// TIA Portal V17 export
// export: Created 2024-09-02T12:50:20.1310188Z, ExportSetting WithDefaults, DisplayName Totally Integrated Automation Portal, DisplayVersion V17, DisplayName TIA Portal Openness, DisplayVersion V17, DisplayName TIA Portal Version Control Interface, DisplayVersion V17, DisplayName STEP 7 Professional, DisplayVersion V17, DisplayName STEP 7 Safety, DisplayVersion V17, DisplayName WinCC Professional, DisplayVersion V17
FUNCTION "AnwFC3_FG02_Saving_Status_SLG3_OP70" : Void   // FC1113, LAD
TITLE = Recalculate Moby / Rückberechnen Moby
{ S7_Optimized_Access := 'TRUE' }
AUTHOR : OlegFuehrus
FAMILY : MOBY
NAME : OlegFuehrus
VERSION : 0.1
// stored: AutoNumber false, IsIECCheckEnabled false, SetENOAutomatically false, UDAEnableTagReadback false
   VAR_TEMP
      t_VKE0 : Bool;   // VKE0
      t_VKE1 : Bool;   // VKE1
      t_Melderk_IO : Bool;   // Meldekontrollen SOLL==IST / Reporting controls SOLL==IST
      t_Status : Byte;   // Bearbeitungstatus / Processing status
      t_TafNr : Int;   // Aktuelle TAF Nummer / Current TAF number
      t_BeaNr : Int;   // Aktuelle BEA Nummer / Current BEA number
      t_END : Bool;
      Save_IO : Bool;
      Save_IO_1 : Bool;
   END_VAR
   VAR CONSTANT
      konst_kennung_schrauber : Byte := 31;
      konst_kennung_fuegen : Byte := 42;
      konst_kennung_wegmessung : Byte := 45;
      konst_kennung_reibmoment : Byte := 46;
      konst_kennung_losbrechmoment : Byte := 47;
   END_VAR
BEGIN

REGION Network 1: INIT
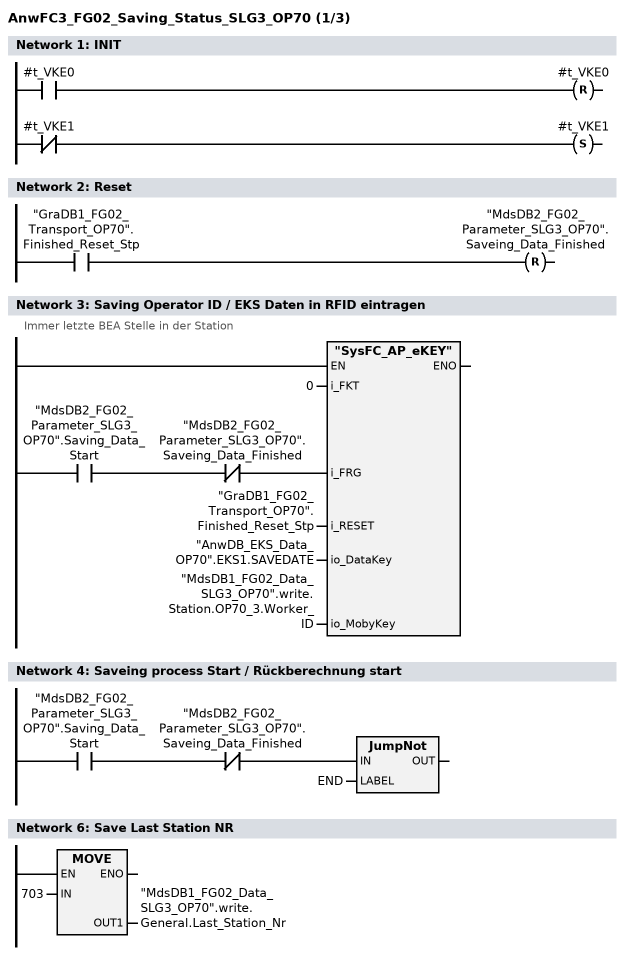
   RUNG wire#powerrail
      Contact( #t_VKE0 )
      R_Coil( #t_VKE0 )
   END_RUNG
   RUNG wire#powerrail
      I_Contact( #t_VKE1 )
      S_Coil( #t_VKE1 )
   END_RUNG
   // the same network as SCL:
   IF #t_VKE0 THEN #t_VKE0 := FALSE; END_IF;
   IF NOT #t_VKE1 THEN #t_VKE1 := TRUE; END_IF;
END_REGION

REGION Network 2: Reset
   RUNG wire#powerrail
      Contact( "GraDB1_FG02_Transport_OP70".Finished_Reset_Stp )
      R_Coil( "MdsDB2_FG02_Parameter_SLG3_OP70".Saveing_Data_Finished )
   END_RUNG
   // the same network as SCL:
   IF "GraDB1_FG02_Transport_OP70".Finished_Reset_Stp THEN
       "MdsDB2_FG02_Parameter_SLG3_OP70".Saveing_Data_Finished := FALSE;
   END_IF;
END_REGION

REGION Network 3: Saving Operator ID / EKS Daten in RFID eintragen
   // Immer letzte BEA Stelle in der Station
   RUNG wire#powerrail
      "SysFC_AP_eKEY"(i_FRG := wire#w1, i_FKT := 0, i_RESET := "GraDB1_FG02_Transport_OP70".Finished_Reset_Stp, io_DataKey := "AnwDB_EKS_Data_OP70".EKS1.SAVEDATE, io_MobyKey := "MdsDB1_FG02_Data_SLG3_OP70".write.Station.OP70_3.Worker_ID)
   END_RUNG
   RUNG wire#powerrail
      Contact( "MdsDB2_FG02_Parameter_SLG3_OP70".Saving_Data_Start )
      I_Contact( "MdsDB2_FG02_Parameter_SLG3_OP70".Saveing_Data_Finished )
   END_RUNG wire#w1
   // the same network as SCL:
   "SysFC_AP_eKEY"(i_FKT := 0,
                   i_FRG := "MdsDB2_FG02_Parameter_SLG3_OP70".Saving_Data_Start AND NOT "MdsDB2_FG02_Parameter_SLG3_OP70".Saveing_Data_Finished,
                   i_RESET := "GraDB1_FG02_Transport_OP70".Finished_Reset_Stp,
                   io_DataKey := "AnwDB_EKS_Data_OP70".EKS1.SAVEDATE,
                   io_MobyKey := "MdsDB1_FG02_Data_SLG3_OP70".write.Station.OP70_3.Worker_ID);
END_REGION

REGION Network 4: Saveing process Start / Rückberechnung start
   // no SCL statement known for JumpNot: written as a call
   JumpNot(in := "MdsDB2_FG02_Parameter_SLG3_OP70".Saving_Data_Start AND NOT "MdsDB2_FG02_Parameter_SLG3_OP70".Saveing_Data_Finished,
           label := END);
END_REGION

REGION Network 5: ################ Status Station / Pallet#################
END_REGION

REGION Network 6: Save Last Station NR
   RUNG wire#powerrail
      Move(in := 703, out1 => "MdsDB1_FG02_Data_SLG3_OP70".write.General.Last_Station_Nr)
   END_RUNG
   // the same network as SCL:
   "MdsDB1_FG02_Data_SLG3_OP70".write.General.Last_Station_Nr := 703;
END_REGION

REGION Network 7: op70 BEA 2 Save Global Status / Status Proces 1
   // IN0 - Aktor ist abgewählt
   // IN1 - TAF ist angewählt
   // IN2 - Nacharbeit in Station
   // IN3 - Auftrag manuell vorgegeben
   // IN4 - Nacharbeit auf Standby-Platz
   // IN5 - Nacharbeit auf EAS-Platz
   // IN6 - TAF hat gearbeitet (Fertigmeldung)
   // IN7 - Bauteil wurde iO bearbeitet
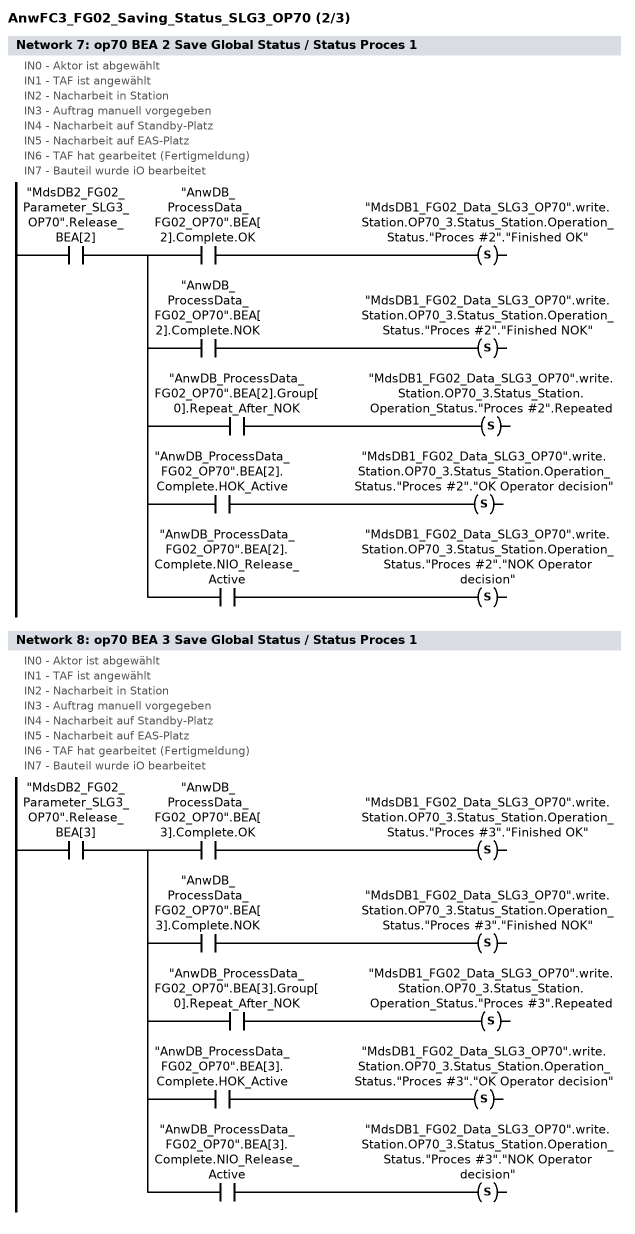
   RUNG wire#powerrail
      Contact( "MdsDB2_FG02_Parameter_SLG3_OP70".Release_BEA[2] )
      wire#w1
      Contact( "AnwDB_ProcessData_FG02_OP70".BEA[2].Complete.OK )
      S_Coil( "MdsDB1_FG02_Data_SLG3_OP70".write.Station.OP70_3.Status_Station.Operation_Status."Proces #2"."Finished OK" )
   END_RUNG
   RUNG wire#w1
      Contact( "AnwDB_ProcessData_FG02_OP70".BEA[2].Complete.NOK )
      S_Coil( "MdsDB1_FG02_Data_SLG3_OP70".write.Station.OP70_3.Status_Station.Operation_Status."Proces #2"."Finished NOK" )
   END_RUNG
   RUNG wire#w1
      Contact( "AnwDB_ProcessData_FG02_OP70".BEA[2].Group[0].Repeat_After_NOK )
      S_Coil( "MdsDB1_FG02_Data_SLG3_OP70".write.Station.OP70_3.Status_Station.Operation_Status."Proces #2".Repeated )
   END_RUNG
   RUNG wire#w1
      Contact( "AnwDB_ProcessData_FG02_OP70".BEA[2].Complete.HOK_Active )
      S_Coil( "MdsDB1_FG02_Data_SLG3_OP70".write.Station.OP70_3.Status_Station.Operation_Status."Proces #2"."OK Operator decision" )
   END_RUNG
   RUNG wire#w1
      Contact( "AnwDB_ProcessData_FG02_OP70".BEA[2].Complete.NIO_Release_Active )
      S_Coil( "MdsDB1_FG02_Data_SLG3_OP70".write.Station.OP70_3.Status_Station.Operation_Status."Proces #2"."NOK Operator decision" )
   END_RUNG
   // the same network as SCL:
   IF "MdsDB2_FG02_Parameter_SLG3_OP70".Release_BEA[2] AND "AnwDB_ProcessData_FG02_OP70".BEA[2].Complete.OK THEN
       "MdsDB1_FG02_Data_SLG3_OP70".write.Station.OP70_3.Status_Station.Operation_Status."Proces #2"."Finished OK" := TRUE;
   END_IF;
   IF "MdsDB2_FG02_Parameter_SLG3_OP70".Release_BEA[2] AND "AnwDB_ProcessData_FG02_OP70".BEA[2].Complete.NOK THEN
       "MdsDB1_FG02_Data_SLG3_OP70".write.Station.OP70_3.Status_Station.Operation_Status."Proces #2"."Finished NOK" := TRUE;
   END_IF;
   IF "MdsDB2_FG02_Parameter_SLG3_OP70".Release_BEA[2] AND "AnwDB_ProcessData_FG02_OP70".BEA[2].Group[0].Repeat_After_NOK THEN
       "MdsDB1_FG02_Data_SLG3_OP70".write.Station.OP70_3.Status_Station.Operation_Status."Proces #2".Repeated := TRUE;
   END_IF;
   IF "MdsDB2_FG02_Parameter_SLG3_OP70".Release_BEA[2] AND "AnwDB_ProcessData_FG02_OP70".BEA[2].Complete.HOK_Active THEN
       "MdsDB1_FG02_Data_SLG3_OP70".write.Station.OP70_3.Status_Station.Operation_Status."Proces #2"."OK Operator decision" := TRUE;
   END_IF;
   IF "MdsDB2_FG02_Parameter_SLG3_OP70".Release_BEA[2] AND "AnwDB_ProcessData_FG02_OP70".BEA[2].Complete.NIO_Release_Active THEN
       "MdsDB1_FG02_Data_SLG3_OP70".write.Station.OP70_3.Status_Station.Operation_Status."Proces #2"."NOK Operator decision" := TRUE;
   END_IF;
END_REGION

REGION Network 8: op70 BEA 3 Save Global Status / Status Proces 1
   // IN0 - Aktor ist abgewählt
   // IN1 - TAF ist angewählt
   // IN2 - Nacharbeit in Station
   // IN3 - Auftrag manuell vorgegeben
   // IN4 - Nacharbeit auf Standby-Platz
   // IN5 - Nacharbeit auf EAS-Platz
   // IN6 - TAF hat gearbeitet (Fertigmeldung)
   // IN7 - Bauteil wurde iO bearbeitet
   RUNG wire#powerrail
      Contact( "MdsDB2_FG02_Parameter_SLG3_OP70".Release_BEA[3] )
      wire#w1
      Contact( "AnwDB_ProcessData_FG02_OP70".BEA[3].Complete.OK )
      S_Coil( "MdsDB1_FG02_Data_SLG3_OP70".write.Station.OP70_3.Status_Station.Operation_Status."Proces #3"."Finished OK" )
   END_RUNG
   RUNG wire#w1
      Contact( "AnwDB_ProcessData_FG02_OP70".BEA[3].Complete.NOK )
      S_Coil( "MdsDB1_FG02_Data_SLG3_OP70".write.Station.OP70_3.Status_Station.Operation_Status."Proces #3"."Finished NOK" )
   END_RUNG
   RUNG wire#w1
      Contact( "AnwDB_ProcessData_FG02_OP70".BEA[3].Group[0].Repeat_After_NOK )
      S_Coil( "MdsDB1_FG02_Data_SLG3_OP70".write.Station.OP70_3.Status_Station.Operation_Status."Proces #3".Repeated )
   END_RUNG
   RUNG wire#w1
      Contact( "AnwDB_ProcessData_FG02_OP70".BEA[3].Complete.HOK_Active )
      S_Coil( "MdsDB1_FG02_Data_SLG3_OP70".write.Station.OP70_3.Status_Station.Operation_Status."Proces #3"."OK Operator decision" )
   END_RUNG
   RUNG wire#w1
      Contact( "AnwDB_ProcessData_FG02_OP70".BEA[3].Complete.NIO_Release_Active )
      S_Coil( "MdsDB1_FG02_Data_SLG3_OP70".write.Station.OP70_3.Status_Station.Operation_Status."Proces #3"."NOK Operator decision" )
   END_RUNG
   // the same network as SCL:
   IF "MdsDB2_FG02_Parameter_SLG3_OP70".Release_BEA[3] AND "AnwDB_ProcessData_FG02_OP70".BEA[3].Complete.OK THEN
       "MdsDB1_FG02_Data_SLG3_OP70".write.Station.OP70_3.Status_Station.Operation_Status."Proces #3"."Finished OK" := TRUE;
   END_IF;
   IF "MdsDB2_FG02_Parameter_SLG3_OP70".Release_BEA[3] AND "AnwDB_ProcessData_FG02_OP70".BEA[3].Complete.NOK THEN
       "MdsDB1_FG02_Data_SLG3_OP70".write.Station.OP70_3.Status_Station.Operation_Status."Proces #3"."Finished NOK" := TRUE;
   END_IF;
   IF "MdsDB2_FG02_Parameter_SLG3_OP70".Release_BEA[3] AND "AnwDB_ProcessData_FG02_OP70".BEA[3].Group[0].Repeat_After_NOK THEN
       "MdsDB1_FG02_Data_SLG3_OP70".write.Station.OP70_3.Status_Station.Operation_Status."Proces #3".Repeated := TRUE;
   END_IF;
   IF "MdsDB2_FG02_Parameter_SLG3_OP70".Release_BEA[3] AND "AnwDB_ProcessData_FG02_OP70".BEA[3].Complete.HOK_Active THEN
       "MdsDB1_FG02_Data_SLG3_OP70".write.Station.OP70_3.Status_Station.Operation_Status."Proces #3"."OK Operator decision" := TRUE;
   END_IF;
   IF "MdsDB2_FG02_Parameter_SLG3_OP70".Release_BEA[3] AND "AnwDB_ProcessData_FG02_OP70".BEA[3].Complete.NIO_Release_Active THEN
       "MdsDB1_FG02_Data_SLG3_OP70".write.Station.OP70_3.Status_Station.Operation_Status."Proces #3"."NOK Operator decision" := TRUE;
   END_IF;
END_REGION

REGION Network 9: op70 Saveing Gobal NOK Status of palet
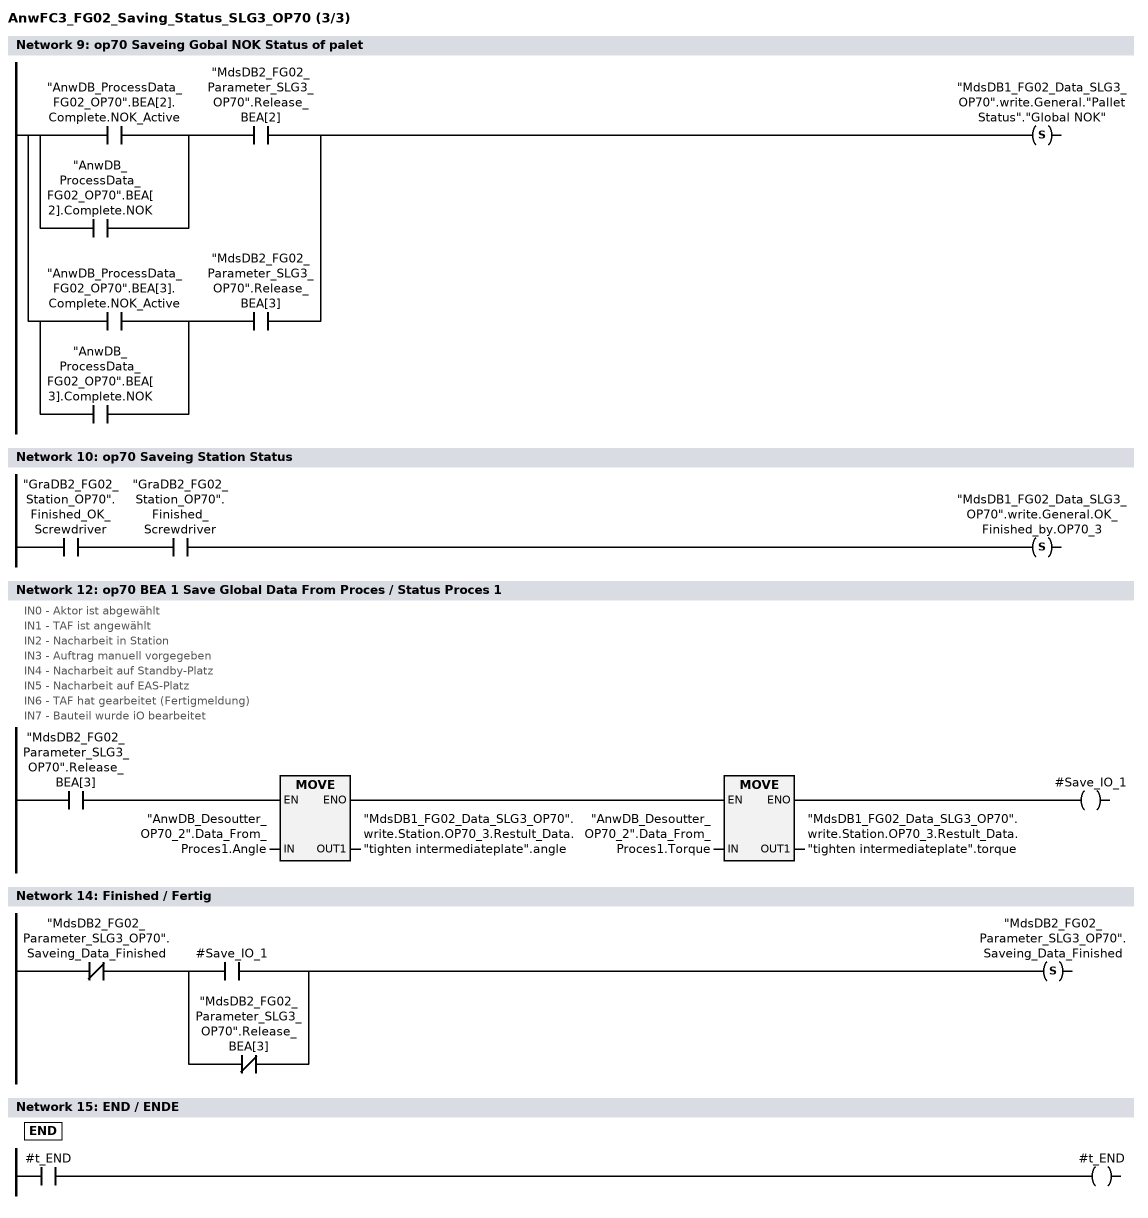
   RUNG wire#powerrail
      Contact( "AnwDB_ProcessData_FG02_OP70".BEA[2].Complete.NOK_Active )
      wire#w1
      Contact( "MdsDB2_FG02_Parameter_SLG3_OP70".Release_BEA[2] )
      wire#w2
      S_Coil( "MdsDB1_FG02_Data_SLG3_OP70".write.General."Pallet Status"."Global NOK" )
   END_RUNG
   RUNG wire#powerrail
      Contact( "AnwDB_ProcessData_FG02_OP70".BEA[2].Complete.NOK )
   END_RUNG wire#w1
   RUNG wire#powerrail
      Contact( "AnwDB_ProcessData_FG02_OP70".BEA[3].Complete.NOK_Active )
      wire#w3
      Contact( "MdsDB2_FG02_Parameter_SLG3_OP70".Release_BEA[3] )
   END_RUNG wire#w2
   RUNG wire#powerrail
      Contact( "AnwDB_ProcessData_FG02_OP70".BEA[3].Complete.NOK )
   END_RUNG wire#w3
   // the same network as SCL:
   IF (("AnwDB_ProcessData_FG02_OP70".BEA[2].Complete.NOK_Active OR "AnwDB_ProcessData_FG02_OP70".BEA[2].Complete.NOK) AND "MdsDB2_FG02_Parameter_SLG3_OP70".Release_BEA[2]) OR (("AnwDB_ProcessData_FG02_OP70".BEA[3].Complete.NOK_Active OR "AnwDB_ProcessData_FG02_OP70".BEA[3].Complete.NOK) AND "MdsDB2_FG02_Parameter_SLG3_OP70".Release_BEA[3]) THEN
       "MdsDB1_FG02_Data_SLG3_OP70".write.General."Pallet Status"."Global NOK" := TRUE;
   END_IF;
END_REGION

REGION Network 10: op70 Saveing Station Status
   RUNG wire#powerrail
      Contact( "GraDB2_FG02_Station_OP70".Finished_OK_Screwdriver )
      Contact( "GraDB2_FG02_Station_OP70".Finished_Screwdriver )
      S_Coil( "MdsDB1_FG02_Data_SLG3_OP70".write.General.OK_Finished_by.OP70_3 )
   END_RUNG
   // the same network as SCL:
   IF "GraDB2_FG02_Station_OP70".Finished_OK_Screwdriver AND "GraDB2_FG02_Station_OP70".Finished_Screwdriver THEN
       "MdsDB1_FG02_Data_SLG3_OP70".write.General.OK_Finished_by.OP70_3 := TRUE;
   END_IF;
END_REGION

REGION Network 11: ################ PROCES DATA ######################
END_REGION

REGION Network 12: op70 BEA 1 Save Global Data From Proces / Status Proces 1
   // IN0 - Aktor ist abgewählt
   // IN1 - TAF ist angewählt
   // IN2 - Nacharbeit in Station
   // IN3 - Auftrag manuell vorgegeben
   // IN4 - Nacharbeit auf Standby-Platz
   // IN5 - Nacharbeit auf EAS-Platz
   // IN6 - TAF hat gearbeitet (Fertigmeldung)
   // IN7 - Bauteil wurde iO bearbeitet
   RUNG wire#powerrail
      Contact( "MdsDB2_FG02_Parameter_SLG3_OP70".Release_BEA[3] )
      Move(in := "AnwDB_Desoutter_OP70_2".Data_From_Proces1.Angle, out1 => "MdsDB1_FG02_Data_SLG3_OP70".write.Station.OP70_3.Restult_Data."tighten intermediateplate".angle)
      Move(in := "AnwDB_Desoutter_OP70_2".Data_From_Proces1.Torque, out1 => "MdsDB1_FG02_Data_SLG3_OP70".write.Station.OP70_3.Restult_Data."tighten intermediateplate".torque)
      Coil( #Save_IO_1 )
   END_RUNG
   // the same network as SCL:
   IF "MdsDB2_FG02_Parameter_SLG3_OP70".Release_BEA[3] THEN
       "MdsDB1_FG02_Data_SLG3_OP70".write.Station.OP70_3.Restult_Data."tighten intermediateplate".angle := "AnwDB_Desoutter_OP70_2".Data_From_Proces1.Angle;
       "MdsDB1_FG02_Data_SLG3_OP70".write.Station.OP70_3.Restult_Data."tighten intermediateplate".torque := "AnwDB_Desoutter_OP70_2".Data_From_Proces1.Torque;
   END_IF;
   #Save_IO_1 := "MdsDB2_FG02_Parameter_SLG3_OP70".Release_BEA[3];
END_REGION

REGION Network 13: ###############################################
END_REGION

REGION Network 14: Finished / Fertig
   RUNG wire#powerrail
      I_Contact( "MdsDB2_FG02_Parameter_SLG3_OP70".Saveing_Data_Finished )
      wire#w1
      Contact( #Save_IO_1 )
      wire#w2
      S_Coil( "MdsDB2_FG02_Parameter_SLG3_OP70".Saveing_Data_Finished )
   END_RUNG
   RUNG wire#w1
      I_Contact( "MdsDB2_FG02_Parameter_SLG3_OP70".Release_BEA[3] )
   END_RUNG wire#w2
   // the same network as SCL:
   IF NOT "MdsDB2_FG02_Parameter_SLG3_OP70".Saveing_Data_Finished AND (#Save_IO_1 OR NOT "MdsDB2_FG02_Parameter_SLG3_OP70".Release_BEA[3]) THEN
       "MdsDB2_FG02_Parameter_SLG3_OP70".Saveing_Data_Finished := TRUE;
   END_IF;
END_REGION

REGION Network 15: END / ENDE
   Label( END )
   RUNG wire#powerrail
      Contact( #t_END )
      Coil( #t_END )
   END_RUNG
   // the same network as SCL:
   END:
   #t_END := #t_END;
END_REGION
END_FUNCTION
